PROGRAM MAIN
VAR
	
	fbPayloadA : Payload_A;
	pPayloadA : POINTER TO Payload_A;
	fbPayloadB : Payload_B;
	fbPayloadCarrier : Payload_Carrier;
	rPayloadAReceiver : REFERENCE TO Payload_A;
	pPayloadAReceiver : POINTER TO Payload_A;
	fbPayloadAReceiver : Payload_A;
	pPayloadBReceiver : POINTER TO Payload_B;
	iPayload : I_Payload;
	step : INT;
	
END_VAR

fbPayloadCarrier();
fbPayloadA();
fbPayloadB();

CASE step OF
	
	1:
	
		IF 	fbPayloadCarrier.SetPayload(fbPayloadA,PAYLOAD_A,ONE_TO_ONE)
			THEN
			
			step := 2;
		END_IF
		
	2:
	
		IF	fbPayloadCarrier.GetPayload(pPayloadAReceiver,PAYLOAD_A)
			THEN
			
			step := 3;
		END_IF
		
	3:
	
	4:

		fbPayloadCarrier.ResetPayload();
		
	10:
	
		pPayloadA := __NEW(PAYLOAD_A);
		IF 	fbPayloadCarrier.SetPayload(pPayloadA^,PAYLOAD_A,ONE_TO_ONE)
			THEN
			
			step := 11;
		END_IF
		
	11:
	
		IF	fbPayloadCarrier.GetPayload(pPayloadAReceiver,PAYLOAD_A)
			THEN
			
			step := 12;
		END_IF
		
	12:
	
	13:
	
		__DELETE(pPayloadA);
		step := 14;
		
	14:
		
	15:

		fbPayloadCarrier.ResetPayload();	
		
END_CASE

END_PROGRAM

(* stored: Version 1.1.0.1, ProductVersion 3.1.4024.2
   POU MAIN: Id {6ebdcdb5-2ed2-420e-97ac-78bc266c18cf}, SpecialFunc None *)
